Staubli VAL3: pallet_setPos.pgx

program pallet_setPos(string x_sPalletName (dimensions=1), num x_nPos (dimensions=1))
begin
  // set the position of the x_sPalletName to x_nPos
  call pallet:setPalletPos(x_sPalletName,x_nPos)
end
